TYPE ST_System_Ampel_Zustand :
STRUCT
	Regelung_Sollw			: ST_System_Ampel_Signal;

	In_Ordnung			: BOOL;

	Stellung : ST_System_Ampel_Signal;
END_STRUCT
END_TYPE

(* stored: Version 1.1.0.1, ProductVersion 3.1.4024.9
   DUT ST_System_Ampel_Zustand: Id {289231fa-2448-460b-a8f5-c259be0ec7a9} *)
